// TIA Portal V19 export
VAR_GLOBAL   // PLC tag table "Straightener_IO"
   Straightener_LiftEntry_V_Close AT %Q131.1 : Bool;   // 836YV2
   Straightener_LiftEntry_V_Open AT %Q131.0 : Bool;   // 836YV1
   Straightener_MotorFan_FdbkKM AT %I3.6 : Bool;   // 832KM1
   Straightener_MotorFan_KM AT %Q1.3 : Bool;   // 832QF1
   Raddrizzatrice_Ls_Rullo_Aperto AT %I129.5 : Bool;   // 836SQ1
   Raddrizzatrice_Phc_Uscita_Prima_Taglio AT %I129.6 : Bool;   // 837BF1
   Raddrizzatrice_Phc_Uscita_Prima_Encoder AT %I129.7 : Bool;   // 837BF2
   Aspo_Phc_Fine_Materiale_Ganasce AT %I126.6 : Bool;   // 736 - LIBERO
   Aspo_Phc_Fine_Materiale_Ing_Raddrizza AT %I126.7 : Bool;   // 736BF2
END_VAR
